(* IEC 61131-3 sources: plc-agent/tests/fixtures/p3_multi/src, 5 files *)

(* ---- Globals.st ---- *)
VAR_GLOBAL
    SystemReady : BOOL := TRUE;
END_VAR

(* ---- FC_Scale.st ---- *)
FUNCTION FC_Scale : REAL
VAR_INPUT
    InputValue : REAL;
END_VAR
FC_Scale := InputValue * 2.0;
END_FUNCTION

(* ---- FB_Alarm.st ---- *)
FUNCTION_BLOCK FB_Alarm
VAR_INPUT
    Trip : BOOL;
END_VAR
VAR_OUTPUT
    Active : BOOL;
END_VAR
Active := Trip;
END_FUNCTION_BLOCK

(* ---- FB_Motor.st ---- *)
FUNCTION_BLOCK FB_Motor
VAR_INPUT
    Start : BOOL;
    Stop : BOOL;
END_VAR
VAR_OUTPUT
    Running : BOOL;
END_VAR
Running := Start AND NOT Stop;
END_FUNCTION_BLOCK

(* ---- Main.st ---- *)
PROGRAM MAIN
VAR
    StartPB AT %IX0.0 : BOOL;
    StopPB AT %IX0.1 : BOOL;
    FaultPB AT %IX0.2 : BOOL;
    Motor AT %QX0.0 : BOOL;
    AlarmOutput AT %QX0.1 : BOOL;
    MotorController : FB_Motor;
    AlarmController : FB_Alarm;
    Scaled : REAL;
END_VAR
MotorController(Start := StartPB, Stop := StopPB);
AlarmController(Trip := FaultPB);
Scaled := FC_Scale(1.0);
Motor := MotorController.Running AND SystemReady;
AlarmOutput := AlarmController.Active;
END_PROGRAM
